// TIA Portal V20 export
// export: Created 2025-12-01T14:57:21.2090707Z, ExportSetting None, DisplayName Totally Integrated Automation Portal, DisplayVersion V20 Update 3, DisplayName TIA Portal Openness, DisplayVersion V20 Update 3, DisplayName TIA Portal Version Control Interface, DisplayVersion V20 Update 3, DisplayName STEP 7 Professional, DisplayVersion V20 Update 3, DisplayName STEP 7 Safety, DisplayVersion V20 Update 2, DisplayName WinCC Basic/Comfort/Advanced, DisplayVersion V20 Update 3, DisplayName WinCC Professional, DisplayVersion V20 Update 3, DisplayName WinCC Unified, DisplayVersion V20 Update 3
DATA_BLOCK "DB2143_DB_STV1"   // DB2140, F_DB
// stored: AutoNumber false, InstanceOfName FB2143_F_Control_STV, InstanceOfType FB
"FB2143_F_Control_STV"
   // VAR_INPUT
   //    NumArmario : Int;
   //    NumLinea : Int;
   //    Desconectar : Bool;
   //    ACK : Bool;
   //    Setas_OK : Bool;
   //    Error_Protusion : Bool;
   //    Barreras_OK : Bool;
   //    Incendio_OK : Bool;
   //    FeedbackPotencia : Bool;
   //    FeedbackFaseRS : Bool;
   //    QBAD_Potencia : Bool;
   //    QBAD_FaseRS : Bool;
   //    ProteccionPotencia : Bool;
   //    ProteccionFaseRS : Bool;
   //    PuertasSect_Abiertas : Bool;
   //    DFK_FireShutterCloseOK : Bool;
   //    DFK_STV_All_Stop : Bool;
   //    PuertasAcceso_Cerradas : Bool;
   //    Vigilancia_PuertasAcceso : Bool;
   // END_VAR
   // VAR_OUTPUT
   //    DFK_Load_Protrusion : Bool;
   //    DFK_Fire_Alarm : Bool;
   //    DFK_FireShutter_Open : Bool;
   //    Cerrar_Puertas_OK : Bool;
   //    Fases_RS_STV : Bool;
   //    Potencia_STV : Bool;
   //    Error_Potencia : Bool;
   //    Error_FaseRS : Bool;
   //    ACK_Next : Bool;
   // END_VAR
   // VAR
   //    MA_DFK_FireShutter_Open : Bool;
   //    MA_Cerrar_Puertas_OK : Bool;
   //    FB_Potencia_STV { S7_SetPoint := 'True'} : "FB2131_F_Linea_Potencia";
   //    FB_Feedback_FaseRS { S7_SetPoint := 'True'} : FDBACK;
   // END_VAR
BEGIN
END_DATA_BLOCK
